ORGANIZATION_BLOCK MAIN:OB1
TITLE=PROGRAM COMMENTS
BEGIN
Network 1 // Network Title
// Network Comment
LD     I0.2
LD     I0.3
LD     I0.0
CTUD   C0, 4
Network 2
LD     I0.0
S      Q0.1, 1
Network 3
LD     I0.0
S      Q0.0, 1
Network 4
LD     I0.1
R      Q0.0, 1
Network 5
LD     I0.1
R      Q0.1, 1
Network 6
LD     C0
R      Q0.0, 1
Network 7
LD     C0
S      Q0.2, 1
Network 8
LD     I0.1
S      Q0.2, 1
Network 9
LD     I0.0
R      Q0.2, 1
Network 10
LD     C0
R      Q0.1, 1
END_ORGANIZATION_BLOCK
SUBROUTINE_BLOCK SBR_0:SBR0
TITLE=SUBROUTINE COMMENTS
BEGIN
Network 1 // Network Title
// Network Comment
END_SUBROUTINE_BLOCK
INTERRUPT_BLOCK INT_0:INT0
TITLE=INTERRUPT ROUTINE COMMENTS
BEGIN
Network 1 // Network Title
// Network Comment
END_INTERRUPT_BLOCK
